(*
 *****************************************************************************
 * timeGetAbsoluteDcTime: Adjust DC time based on the external time signal
 *
 *  IN   ptptime    : External time signal
 *  IN   leapSecond : Leap Second 
 *  OUT  dcTIME     : Adjusted TwinCAT DC time
 ***************************************************************************** 
 *)
FUNCTION F_timeGetAbsoluteDcTime : BOOL
VAR_INPUT
	ptptime:			T_ASTRO_EL6688_DATA;
	nLeapSecond:		DINT;
	DcToExtTimeOffset:	LINT;
END_VAR
VAR_IN_OUT
	dcTime:   ULINT;
END_VAR
VAR
	val:		LINT	:= 0;
	diff:		LINT	:= 0;
	one_sec:	LINT	:= 1000000000;
END_VAR

(*
HRESULT timeGetAbsoluteDcTime(PTPTime ptptime, INT leapSecond, LONGLONG *dcTime)
{
	HRESULT hr = S_OK; 
	LONGLONG val = 0;
	LONGLONG diff = 0;
	LONGLONG ONE_SEC = 1000000000;
	
	// Check if external time signal is connected
	if (ptptime.not_connected)
		return S_FALSE;

	// If both variables are null means most probably they are not mapped.
	if (ptptime.internal == 0 || ptptime.external == 0)
		return S_FALSE;

	diff = (ptptime.internal - ptptime.external) + (ONE_SEC * leapSecond) + ptptime.dcTcOffset;
	*dcTime -=  diff;
	return hr;
}*)

// Check if external time signal is connected
IF ptptime.External_device_not_connected THEN
	F_timeGetAbsoluteDcTime := FALSE;
END_IF

// If both variables are null means most probably they are not mapped.
// TODO: Is it OR or AND ?
IF ptptime.Internal_time_stamp = 0  OR  ptptime.External_time_stamp = 0 THEN
	F_timeGetAbsoluteDcTime := FALSE;
END_IF

diff := (ULINT_TO_LINT(ptptime.Internal_time_stamp) - ULINT_TO_LINT(ptptime.External_time_stamp)) + 
		(one_sec * nLeapSecond) + DcToExtTimeOffset;

dcTime	:= dcTime - LINT_TO_ULINT(diff);

F_timeGetAbsoluteDcTime := TRUE;

END_FUNCTION

(* stored: Version 1.1.0.1, ProductVersion 3.1.4022.9
   POU F_timeGetAbsoluteDcTime: Id {6a13050b-7de1-4074-8d3e-b4d423a6ff66}, SpecialFunc None *)
